(* CoDeSys 2.3 export: FK16PUMPSFAULTYCONTROL.EXP *)

(* POU K16/fK16PumpsFaultyControl, ST *)
FUNCTION fK16PumpsFaultyControl :BOOL
(* Проверка состояния насосов*)
VAR_INPUT
	PumpState : ARRAY [1..MAX_K16_PUMPS_NUM] OF BOOL;
	PumpStatusCheckDelay : ARRAY [1..MAX_K16_PUMPS_NUM] OF BOOL;
	PressureDrop : BOOL;
END_VAR
VAR
	i : USINT;
	activePumpID : USINT; (*номер работающего насоса*)
END_VAR
activePumpID := 0;

FOR i := 1 TO MAX_K16_PUMPS_NUM DO
	IF PumpState[i] THEN
		IF activePumpID <> 0 THEN
			(*
				Включено больше одного насоса -
				ничего не можем сказать об их исправности
			*)
			RETURN;
		END_IF;
		activePumpID := i;
	END_IF;
END_FOR;

IF activePumpID = 0 THEN
	(*
		Не включен ни один насос - 
		ничего не можем сказать об их исправности
	*)
	RETURN;
END_IF;

IF PumpStatusCheckDelay[activePumpID] THEN
	(*
		Определяем исправность насоса
		по перепаду давления
	*)
	K16PumpFaulty[activePumpID] := NOT(PressureDrop);
END_IF;
END_FUNCTION
